Staubli VAL3: cmdQuickStop.pgx

public program cmdQuickStop(num x_nAxNum)
begin
  //"quickstop"置为false
  //激活quickstop
  if !bQuickStop[x_nAxNum]
    doFaultReset[x_nAxNum]=false
    doEnableVoltage[x_nAxNum]=true
    doSwitchOn[x_nAxNum]=true
    doEnableOp[x_nAxNum]=true
    delay(0.1)
    doQuickStop[x_nAxNum]=false
    delay(0.1)
  endIf
end
